// TwinCAT 3 PLC project Untitled1
// ProgramVersion: 3.1.4024.0
// libraries:
//   Tc2_Standard, * (Beckhoff Automation GmbH)
//   Tc2_System, * (Beckhoff Automation GmbH)
//   Tc3_Module, * (Beckhoff Automation GmbH)
//   VisuDialogs, * (System)
// project tree:
//   DUTs/ ST_robot.TcDUT
//   / GlobalTextList.TcGTLO, PlcTask.TcTTO, Visualization Manager.TcVMO (not stored)
//   GVLs/ GVL.TcGVL
//   POUs/ FBDsRULE.TcPOU, MAIN.TcPOU, POU.TcPOU
//   VISUs/ Visualization.TcVIS
// real-time tasks:
//   TASK PlcTask: cycle T#10ms, priority 20, ADS port 350

CONFIGURATION Untitled1
    RESOURCE PLC ON TwinCAT3
        TASK PlcTask(INTERVAL := T#10ms, PRIORITY := 20);
        PROGRAM MAIN WITH PlcTask : MAIN;
    END_RESOURCE
END_CONFIGURATION

// ---- DUTs/ST_robot.TcDUT
TYPE ST_robot :
STRUCT
	Xstatus: BOOL;
	rTemp: REAL;
	aDirection: ARRAY [1..4] OF BOOL;
END_STRUCT
END_TYPE

// ---- GVLs/GVL.TcGVL
{attribute 'Tc2GvlVarNames'}
VAR_GLOBAL
	button : BOOL;
	
	light1: BOOL;
	light2: BOOL;
	light3: BOOL;
	light4: BOOL;
	
	alights: ARRAY[1..4] OF BOOL;
	Hold : INT;
	
	NUM : INT;
    CAS: INT ;
	
	robo1 : ST_robot; 
	robo2 : ST_robot;
	
	test: bool;
END_VAR

// ---- POUs/MAIN.TcPOU
PROGRAM MAIN
VAR
	VarTest1: BOOL;
	UmpaLumpa: BOOL;
END_VAR

FOR hold := 1 TO 4 DO
	aLIghts[hold] := FALSE;
END_FOR

CASE CAS OF	
	0, 5..8:
	
		IF (NUM > 0) AND (NUM < 100) THEN;
			alights[1] := TRUE;
		
		ELSIF (NUM > 101) AND (NUM < 200) THEN;
			alights[2] := TRUE;
		END_IF
		
	1,2,3,4:
	
		IF (NUM > 201) AND (NUM < 300) THEN;
			alights[3] := TRUE;
		
		ELSIF (NUM > 301) AND (NUM < 400) THEN;
			alights[4] := TRUE;
			
		END_IF	
	
END_CASE
	
IF test := TRUE THEN;
	robo1.aDirection[1] := TRUE;
	
	robo2.aDirection[3] := TRUE;
END_IF


POU();


//adding things to this is fun

VarTest1 := TRUE;


UmpaLumpa := FALSE;

END_PROGRAM

// ---- POUs/POU.TcPOU
PROGRAM POU
VAR
	Ton1 :ton;
	Ton2 :ton;
	
END_VAR


ton1(PT := T#2S);
ton2(PT := T#2S);


IF ton2.Q = TRUE THEN
			ton1.in :=FALSE;
			ton2.IN :=FALSE;
			
ELSIF ton1.Q = TRUE THEN
		ton2.IN := TRUE;
				
ELSIF ton2.Q = FALSE THEN
	ton1.IN := TRUE;
	
	
END_IF

END_PROGRAM

// ---- POUs/FBDsRULE.TcPOU
PROGRAM FBDsRULE
VAR
	nothingspecial : BOOL;
	
END_VAR

// NETWORK 1

END_PROGRAM

// ---- GlobalTextList.TcGTLO
TEXTLIST GlobalTextList
  967 = '%d'
  185 = 'CASE Ranges'
  445 = 'Hello'
  54 = 'IF ranges'
END_TEXTLIST

// ---- VISUs/Visualization.TcVIS
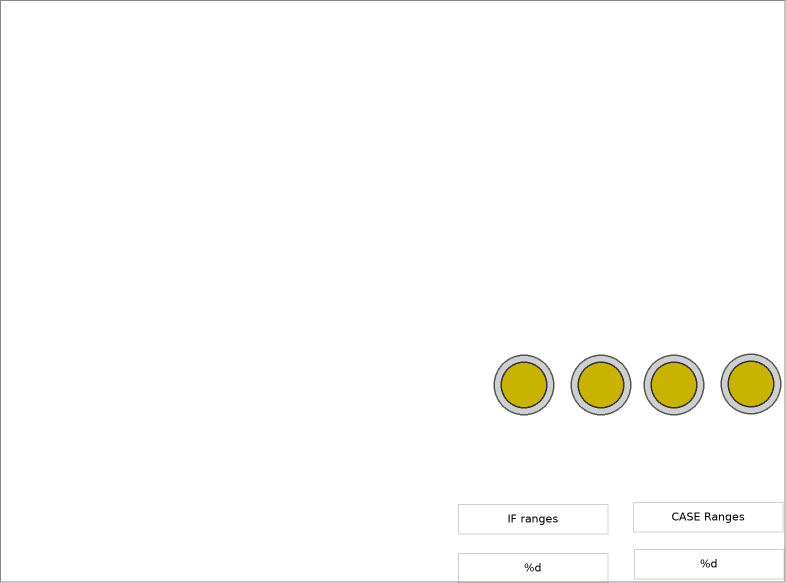
VISUALIZATION Visualization  // 786x583
    Lamp1 (489,350 70x70), variable: alights[1], style: Lamp-Lamp1-Yellow
    Textfield (458,553 150x30), "%d", text variable: NUM
        OnMouseClick: write the text variable via Edit
    Lamp1 (566,350 70x70), variable: alights[2], style: Lamp-Lamp1-Yellow
    Lamp1 (639,350 70x70), variable: alights[3], style: Lamp-Lamp1-Yellow
    Lamp1 (716,349 70x70), variable: alights[4], style: Lamp-Lamp1-Yellow
    Textfield (458,504 150x30), "IF ranges"
    Textfield (633,502 150x30), "CASE Ranges"
    Textfield (634,549 150x30), "%d", text variable: CAS
        OnMouseClick: write the text variable via Edit
END_VISUALIZATION
